(* IEC 61131-3 sources: programs/VI-54/VI-54_20171205/VI-54_20171205/Stations/Screen/LseClass170718/Class/PlcOnline, 1 file *)

(* ---- PlcOnline.st ---- *)
(*!
<Class
	Name               = "PlcOnline"
	Revision           = "0.0"
	RealtimeTask       = "false"
	CyclicTask         = "false"
	BackgroundTask     = "true"
	Sigmatek           = "false"
	OSInterface        = "false"
	HighPriority       = "false"
	Automatic          = "false"
	UpdateMode         = "Prescan"
	SharedCommandTable = "true"
	Objectsize         = "(570,120)">
	<Channels>
		<Server Name="ClassSvr" Visualized="false" Initialize="false" WriteProtected="true" Retentive="false"/>
		<Server Name="WindowNbr" Visualized="false" Initialize="true" WriteProtected="true" Retentive="false"/>
		<Client Name="ActWindow" Required="true" Internal="false"/>
		<Client Name="LogOut" Required="true" Internal="false"/>
	</Channels>
</Class>
*)
PlcOnline : CLASS
  //Servers:
	ClassSvr 	: SvrChCmd_DINT;
	WindowNbr 	: SvrCh_DINT;
  //Clients:
	ActWindow 	: CltCh_DINT;
	LogOut 	: CltCh_DINT;
  //Variables:
		OldWindow 	: DINT;
  //Functions:

	FUNCTION VIRTUAL GLOBAL Background
		VAR_INPUT
			EAX 	: UDINT;
		END_VAR
		VAR_OUTPUT
			state (EAX) 	: UDINT;
		END_VAR;
  //Tables:
	FUNCTION @STD
		VAR_OUTPUT
			ret_code	: CONFSTATES;
		END_VAR;
	FUNCTION GLOBAL TAB @CT_;
END_CLASS;

FUNCTION VIRTUAL GLOBAL PlcOnline::Background
	VAR_INPUT
		EAX 	: UDINT;
	END_VAR
	VAR_OUTPUT
		state (EAX) 	: UDINT;
	END_VAR

  // Read act window
  ActWindow := ActWindow.Read();

  // Log out automatically

  if OldWindow <> ActWindow then
    if ActWindow = WindowNbr then
      LogOut.Write(input:= 5);
    end_if;
    OldWindow := ActWindow;
  end_if;

	state := READY;

END_FUNCTION
